{attribute addProperty BoxType "EL9930-0000-0016"}
{attribute addProperty Id "A_0002_EL9930_0001_0016EL9930_56E76016182.25A_0003_EL9930_0000_0017A_0003_EL9930_0000_0017_255119B7182.25"}
{attribute addProperty CRC "2181094320"}
{attribute addProperty SizeInBites "36"}
{attribute addProperty SizeInBytes "4.5"}
TYPE A_0001_EL9930_0000_0016_8200DBB0 EXTENDS EL9930_A7E0D8F4 :
STRUCT
	{attribute addProperty Name "A_0002_EL9930_0001_0016"}
	A_0002_EL9930_0001_0016 : EL9930_56E76016;
	{attribute addProperty Name "A_0003_EL9930_0000_0017"}
	A_0003_EL9930_0000_0017 : A_0003_EL9930_0000_0017_255119B7;
END_STRUCT
END_TYPE

(* stored: Version 1.2.0.0, ProductVersion 3.1.4024.9
   DUT A_0001_EL9930_0000_0016_8200DBB0: Id {4097eb44-3602-4869-8c6d-d94998b7ec36} *)
